// Mitsubishi GX Works2 project: 금속비금속 터치스크린   PLC: Q02/Q02H

PROGRAM MAIN
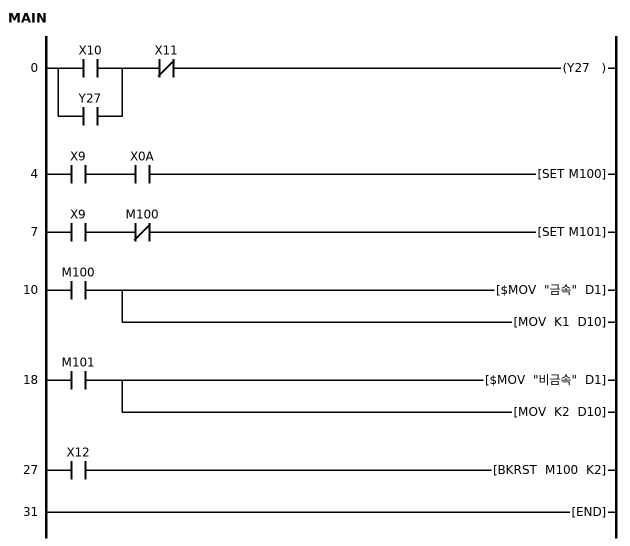
0     LD      X10
      OR      Y27
      ANI     X11
      OUT     Y27
4     LD      X9
      AND     X0A
      SET     M100
7     LD      X9
      ANI     M100
      SET     M101
10    LD      M100
      $MOV    "금속" D1
      MOV     K1 D10
18    LD      M101
      $MOV    "비금속" D1
      MOV     K2 D10
27    LD      X12
      BKRST   M100 K2
31    END
END_PROGRAM
